Fanuc KAREL source: kb00094.KL

-- PROVISIONAL review KL for V1013-1; original PC SHA256 f068cc674cc5b2009233c340b4a3a749f40abb91c8bf6e328367841815c06ab1
-- Incomplete behavior may be omitted. Consult companion uncertainty JSON. Do not deploy.
PROGRAM KB00094
%NOLOCKGROUP
BEGIN
  -- UNRESOLVED_PC offsets 5-12; opcodes 9D,23
  -- UNRESOLVED_PC offsets 17-27; opcodes 27,22,31
  -- UNRESOLVED_PC offsets 32-36; opcodes 7F
END KB00094
